{attribute addProperty BoxType "AMI8000-0000-0016"}
{attribute addProperty Id "PositionAT %I*UDINT324"}
{attribute addProperty CRC "3129649648"}
{attribute addProperty SizeInBites "32"}
{attribute addProperty SizeInBytes "4"}
TYPE FB_Position_BA8AA9F0 :
STRUCT
	{attribute addProperty Name "Position"}
	Position AT %I* : UDINT;
END_STRUCT
END_TYPE

(* stored: Version 1.2.0.0, ProductVersion 3.1.4024.9
   DUT FB_Position_BA8AA9F0: Id {bdf757a2-f6b2-43a7-bb16-9a4f68619ce0} *)
